KUKA KRL program: C2_CicloCompleto.src, C2_CicloCompleto.dat

--- C2_CicloCompleto.src ---
&ACCESS RVO1
&REL 253
&PARAM DISKPATH = KRC:\R1\Program\Work
DEF  C2_CicloCompleto (limpieza:IN)
   BOOL bTornillo, limpieza
   DECL INT velocidadAnterior,contadorPasadasLaser
   ;FOLD PROGRAM INFO --------------------------------------------------------
      ; Program: C2_CicloCompleto
      ; Description:
      ; Creation Date: 16/04/2024
      ; Last Modification Date: 14/09/2025
      ; Author:
      ;           Alexander Kalis
      ;           Tekniker, C. Iñaki Goenaga, 5, 20600, Gipuzkoa
      ;           +34 674 05 15 10
      ;           alexander.kalis@tekniker.es
      ; Last modification Author:
      ;           Alexander Kalis
      ; Customer: Erreka S. COOP
   ;ENDFOLD --------------------------------------------------------

   ;FOLD INI;%{PE}
      ;FOLD BASISTECH INI
         GLOBAL INTERRUPT DECL 3 WHEN $STOPMESS==TRUE DO IR_STOPM ( )
         INTERRUPT ON 3
         BAS (#INITMOV,0 )
      ;ENDFOLD (BASISTECH INI)

      ;FOLD USER INI
         ;Make your modifications here
         bTornillo=$IN[139]
         contadorPasadasLaser=0
         ;laserFrames = posCalcLaserSweep($RECIPE, $LAYOUT)
         ;laserFrames = posCalcLaserSweepAngledP($RECIPE, $LAYOUT, 5)
         laserFrames = posCalcLaserSweepAngledN($RECIPE, $LAYOUT, angle_barrido_laserAB)

         ;paintFrames = posCalcPaintSweep($RECIPE, $LAYOUT)
         ;paintFrames = posCalcPaintSweepAngledP($RECIPE, $LAYOUT, 5)
         paintFrames = posCalcPaintSweepAngledN($RECIPE, $LAYOUT, angle_barrido_pinturaAB)
      ;ENDFOLD (USER INI)
   ;ENDFOLD (INI)

   ;FOLD SPTP HOME CONT Vel=100 % DEFAULT ;%{PE}
      ;FOLD Parameters ;%{h}
         ;Params IlfProvider=kukaroboter.basistech.inlineforms.movement.spline; Kuka.IsGlobalPoint=False; Kuka.PointName=HOME; Kuka.BlendingEnabled=True; Kuka.MoveDataPtpName=DEFAULT; Kuka.VelocityPtp=100; Kuka.VelocityFieldEnabled=True; Kuka.ColDetectFieldEnabled=True; Kuka.CurrentCDSetIndex=0; Kuka.MovementParameterFieldEnabled=True; IlfCommand=SPTP
      ;ENDFOLD
      SPTP XHOME WITH $VEL_AXIS[1] = SVEL_JOINT(100.0), $TOOL = STOOL2(FHOME), $BASE = SBASE(FHOME.BASE_NO), $IPO_MODE = SIPO_MODE(FHOME.IPO_FRAME), $LOAD = SLOAD(FHOME.TOOL_NO), $ACC_AXIS[1] = SACC_JOINT(PDEFAULT), $APO = SAPO_PTP(PDEFAULT), $GEAR_JERK[1] = SGEAR_JERK(PDEFAULT), $COLLMON_TOL_PRO[1] = USE_CM_PRO_VALUES(0) C_Spl
   ;ENDFOLD

   ;FOLD Path to laser station
      IF limpieza THEN
         ;FOLD SPTP PTL1 CONT Vel=100 % PDAT13 Tool[1]:pintxoEstatico Base[2]:laserTCP extTCP  ;%{PE}
            ;FOLD Parameters ;%{h}
               ;Params IlfProvider=kukaroboter.basistech.inlineforms.movement.spline; Kuka.IsGlobalPoint=False; Kuka.PointName=PTL1; Kuka.BlendingEnabled=True; Kuka.MoveDataPtpName=PDAT13; Kuka.VelocityPtp=100; Kuka.VelocityFieldEnabled=True; Kuka.ColDetectFieldEnabled=True; Kuka.CurrentCDSetIndex=0; Kuka.MovementParameterFieldEnabled=True; IlfCommand=SPTP
            ;ENDFOLD
            SPTP XPTL1 WITH $VEL_AXIS[1] = SVEL_JOINT(100.0), $TOOL = STOOL2(FPTL1), $BASE = SBASE(FPTL1.BASE_NO), $IPO_MODE = SIPO_MODE(FPTL1.IPO_FRAME), $LOAD = SLOAD(FPTL1.TOOL_NO), $ACC_AXIS[1] = SACC_JOINT(PPDAT13), $APO = SAPO_PTP(PPDAT13), $GEAR_JERK[1] = SGEAR_JERK(PPDAT13), $COLLMON_TOL_PRO[1] = USE_CM_PRO_VALUES(0) C_Spl
         ;ENDFOLD
   ;ENDFOLD

   ;FOLD LASER PROCESS
      ;FOLD INIT barrido
         $TOOL = TOOL_DATA[1]
         $BASE = BASE_DATA[2]
         $IPO_MODE = #TCP
      ;ENDFOLD

      ;BUCLE DEPENDIENDO DEL NUMERO DE PASADAS

      ;FOLD Limpieza exterior esparrago
         $TOOL = TOOL_DATA[1] : laserFrames.screwBottom
         TRIGGER WHEN PATH = 0 ONSTART DELAY = 0 DO autMotorON() PRIO = 101
         TRIGGER WHEN PATH = 0 ONSTART DELAY = 0 DO autLaserON() PRIO = 102
         SPTP $NULLFRAME:C2LaserOffset[$RECIPE.recipeNum].sBO WITH $VEL.CP = laserParameter[$RECIPE.recipeNum].vel2, $VEL.ORI1 = laserParameter[$RECIPE.recipeNum].velRot2, $VEL.ORI2 = laserParameter[$RECIPE.recipeNum].velRot2
         WAIT SEC laserParameter[$RECIPE.recipeNum].tClean1
      ;ENDFOLD
      ;FOLD Limpieza perfil esparrago (punto A)
         $TOOL = TOOL_DATA[1] : laserFrames.screwProfileA
         SLIN $NULLFRAME:C2LaserOffset[$RECIPE.recipeNum].sPAO WITH $VEL.CP = laserParameter[$RECIPE.recipeNum].vel1, $VEL.ORI1 = laserParameter[$RECIPE.recipeNum].velRot1, $VEL.ORI2 = laserParameter[$RECIPE.recipeNum].velRot1
      ;ENDFOLD
      ;FOLD Limpieza perfil esparrago (punto B)
         velocidadAnterior = $OV_PRO
         $OV_PRO = 100
         $TOOL = TOOL_DATA[1] : laserFrames.screwProfileB
         SLIN $NULLFRAME:C2LaserOffset[$RECIPE.recipeNum].sPBO WITH $VEL.CP = laserParameter[$RECIPE.recipeNum].velSweep, $VEL.ORI1 = laserParameter[$RECIPE.recipeNum].velRot1, $VEL.ORI2 = laserParameter[$RECIPE.recipeNum].velRot1
         $OV_PRO = velocidadAnterior
      ;ENDFOLD
      contadorPasadasLaser=contadorPasadasLaser+1
      IF (bTornillo) THEN
         ;FOLD Limpieza perfil cabeza
            $TOOL = TOOL_DATA[1] : laserFrames.screwHex
            SLIN $NULLFRAME:C2LaserOffset[$RECIPE.recipeNum].sHO WITH $VEL.CP = laserParameter[$RECIPE.recipeNum].vel1, $VEL.ORI1 = laserParameter[$RECIPE.recipeNum].velRot1, $VEL.ORI2 = laserParameter[$RECIPE.recipeNum].velRot1
            WAIT SEC laserParameter[$RECIPE.recipeNum].tHex
         ;ENDFOLD
         ;FOLD Limpieza interior cabeza
            $TOOL = TOOL_DATA[1] : laserFrames.screwInnerHead
            SLIN $NULLFRAME:C2LaserOffset[$RECIPE.recipeNum].sIHO WITH $VEL.CP = laserParameter[$RECIPE.recipeNum].vel1, $VEL.ORI1 = laserParameter[$RECIPE.recipeNum].velRot1, $VEL.ORI2 = laserParameter[$RECIPE.recipeNum].velRot1
            WAIT SEC laserParameter[$RECIPE.recipeNum].tClean2
         ;ENDFOLD
      ENDIF

      ;FOLD Limpieza exterior cabeza
         $TOOL = TOOL_DATA[1] : laserFrames.screwOuterHead
         SLIN $NULLFRAME:C2LaserOffset[$RECIPE.recipeNum].sOHO WITH $VEL.CP = laserParameter[$RECIPE.recipeNum].vel1, $VEL.ORI1 = laserParameter[$RECIPE.recipeNum].velRot1, $VEL.ORI2 = laserParameter[$RECIPE.recipeNum].velRot1
         WAIT SEC laserParameter[$RECIPE.recipeNum].tClean3
      ;ENDFOLD
      ;Vuelta con angulo negativo B->A
      WHILE (ByNPasadasLaser > contadorPasadasLaser)
         ;FOLD Limpieza perfil esparrago (punto B)
            $TOOL = TOOL_DATA[1] : laserFrames.screwProfileB
            SLIN $NULLFRAME:C2LaserOffset[$RECIPE.recipeNum].sPBO WITH $VEL.CP = laserParameter[$RECIPE.recipeNum].vel1, $VEL.ORI1 = laserParameter[$RECIPE.recipeNum].velRot1, $VEL.ORI2 = laserParameter[$RECIPE.recipeNum].velRot1
         ;ENDFOLD
         ;FOLD Limpieza perfil esparrago (punto A)
            $TOOL = TOOL_DATA[1] : laserFrames.screwProfileA
            SLIN $NULLFRAME:C2LaserOffset[$RECIPE.recipeNum].sPAO WITH $VEL.CP = laserParameter[$RECIPE.recipeNum].velSweep, $VEL.ORI1 = laserParameter[$RECIPE.recipeNum].velRot1, $VEL.ORI2 = laserParameter[$RECIPE.recipeNum].velRot1
         ;ENDFOLD
         contadorPasadasLaser = contadorPasadasLaser + 1
      ENDWHILE
      autLaserOFF()
      autMotorOff()
      ENDIF
         ;ENDFOLD


   ;FOLD Path to DRYZONE
      petitionPermission(bPetEntradaLamparas, bPermisoEntradaLamparas)
   ;ENDFOLD

   ;FOLD Path to Paint station
      ;FOLD SPTP LTP1 CONT Vel=100 % PDAT17 Tool[1]:pintxoEstatico Base[3]:pintura ;%{PE}
         ;FOLD Parameters ;%{h}
            ;Params IlfProvider=kukaroboter.basistech.inlineforms.movement.spline; Kuka.IsGlobalPoint=False; Kuka.PointName=LTP1; Kuka.BlendingEnabled=True; Kuka.MoveDataPtpName=PDAT17; Kuka.VelocityPtp=100; Kuka.VelocityFieldEnabled=True; Kuka.ColDetectFieldEnabled=True; Kuka.CurrentCDSetIndex=0; Kuka.MovementParameterFieldEnabled=True; IlfCommand=SPTP
         ;ENDFOLD
         SPTP XLTP1 WITH $VEL_AXIS[1] = SVEL_JOINT(100.0), $TOOL = STOOL2(FLTP1), $BASE = SBASE(FLTP1.BASE_NO), $IPO_MODE = SIPO_MODE(FLTP1.IPO_FRAME), $LOAD = SLOAD(FLTP1.TOOL_NO), $ACC_AXIS[1] = SACC_JOINT(PPDAT17), $APO = SAPO_PTP(PPDAT17), $GEAR_JERK[1] = SGEAR_JERK(PPDAT17), $COLLMON_TOL_PRO[1] = USE_CM_PRO_VALUES(0) C_Spl
      ;ENDFOLD

   ;ENDFOLD

   ;FOLD PAINT PROCESS

      ;FOLD INIT barrido
         $TOOL = TOOL_DATA[1]
         $BASE = BASE_DATA[3]
         $IPO_MODE = #TCP
      ;ENDFOLD

      ;FOLD Pintado exterior esparrago
         TRIGGER WHEN PATH = 0 DELAY = 0 DO autPaintON() PRIO = 108
         TRIGGER WHEN PATH = 0 ONSTART DELAY = 0 DO autMotorOn() PRIO = 109
         $TOOL = TOOL_DATA[1] : paintFrames.screwBottom
         SPTP $NULLFRAME WITH $VEL.CP = paintParameter[$RECIPE.recipeNum].vel2, $VEL.ORI1 = paintParameter[$RECIPE.recipeNum].velRot2, $VEL.ORI2 = paintParameter[$RECIPE.recipeNum].velRot2
         WAIT SEC paintParameter[$RECIPE.recipeNum].tPaint1
         TRIGGER WHEN PATH = 0 ONSTART DELAY = 0 DO autPaintOFF() PRIO = 110
      ;ENDFOLD
      ;FOLD Pintado perfil esparrago (punto A)
         velocidadAnterior = $OV_PRO
         $TOOL = TOOL_DATA[1] : paintFrames.screwProfileA
         TRIGGER WHEN PATH = 0 DELAY = 0 DO autPaintON() PRIO = 111

         SLIN $NULLFRAME WITH $VEL.CP = paintParameter[$RECIPE.recipeNum].vel1, $VEL.ORI1 = paintParameter[$RECIPE.recipeNum].velRot1, $VEL.ORI2 = paintParameter[$RECIPE.recipeNum].velRot1
         $OV_PRO = 100
      ;ENDFOLD
      ;FOLD Pintado perfil esparrago (punto B)
         $TOOL = TOOL_DATA[1] : paintFrames.screwProfileB
         SLIN $NULLFRAME  WITH $VEL.CP = paintParameter[$RECIPE.recipeNum].velSweep, $VEL.ORI1 = paintParameter[$RECIPE.recipeNum].velRot1, $VEL.ORI2 = paintParameter[$RECIPE.recipeNum].velRot1
         TRIGGER WHEN PATH = 0 ONSTART DELAY = 0 DO autPaintOFF() PRIO = 112
         $OV_PRO = velocidadAnterior
      ;ENDFOLD
      IF (bTornillo) THEN
         ;FOLD Pintado perfil cabeza
            $TOOL = TOOL_DATA[1] : paintFrames.screwHex
            SLIN $NULLFRAME  WITH $VEL.CP = paintParameter[$RECIPE.recipeNum].vel1, $VEL.ORI1 = paintParameter[$RECIPE.recipeNum].velRot1, $VEL.ORI2 = paintParameter[$RECIPE.recipeNum].velRot1
            TRIGGER WHEN PATH = 0 DELAY = 0 DO autPaintON() PRIO = 113
            WAIT SEC paintParameter[$RECIPE.recipeNum].tHex
            TRIGGER WHEN PATH = 0 ONSTART DELAY = 0 DO autPaintOFF() PRIO = 114
         ;ENDFOLD
         ;FOLD Pintado interior cabeza
            TRIGGER WHEN PATH = 0 DELAY = 0 DO autPaintON() PRIO = 115
            $TOOL = TOOL_DATA[1] : paintFrames.screwInnerHead
            SLIN $NULLFRAME  WITH $VEL.CP = paintParameter[$RECIPE.recipeNum].vel1, $VEL.ORI1 = paintParameter[$RECIPE.recipeNum].velRot1, $VEL.ORI2 = paintParameter[$RECIPE.recipeNum].velRot1
            WAIT SEC paintParameter[$RECIPE.recipeNum].tPaint2
            TRIGGER WHEN PATH = 0 ONSTART DELAY = 0 DO autPaintOFF() PRIO = 116
         ;ENDFOLD
      ENDIF
      ;FOLD Pintado exterior cabeza
         $TOOL = TOOL_DATA[1] : paintFrames.screwOuterHead
         TRIGGER WHEN PATH = 0 DELAY = 0 DO autPaintON() PRIO = 117
         SPTP $NULLFRAME WITH $VEL.CP = paintParameter[$RECIPE.recipeNum].vel1, $VEL.ORI1 = paintParameter[$RECIPE.recipeNum].velRot1, $VEL.ORI2 = paintParameter[$RECIPE.recipeNum].velRot1
         WAIT SEC paintParameter[$RECIPE.recipeNum].tPaint3
         TRIGGER WHEN PATH = 0 ONSTART DELAY = 0 DO autPaintOFF() PRIO = 118
         autLamaparasOn()
      ;ENDFOLD

   ;ENDFOLD

   dryPos = posCalcDry($RECIPE, $LAYOUT)

   ;FOLD Path to wait Zone
;FOLD SPTP p10 CONT Vel=100 % PDAT19 Tool[1]:pintxoEstatico Base[4]:lamparas ;%{PE}
;FOLD Parameters ;%{h}
;Params IlfProvider=kukaroboter.basistech.inlineforms.movement.spline; Kuka.IsGlobalPoint=False; Kuka.PointName=p10; Kuka.BlendingEnabled=True; Kuka.MoveDataPtpName=PDAT19; Kuka.VelocityPtp=100; Kuka.VelocityFieldEnabled=True; Kuka.ColDetectFieldEnabled=True; Kuka.CurrentCDSetIndex=0; Kuka.MovementParameterFieldEnabled=True; IlfCommand=SPTP
;ENDFOLD
SPTP Xp10 WITH $VEL_AXIS[1] = SVEL_JOINT(100.0), $TOOL = STOOL2(Fp10), $BASE = SBASE(Fp10.BASE_NO), $IPO_MODE = SIPO_MODE(Fp10.IPO_FRAME), $LOAD = SLOAD(Fp10.TOOL_NO), $ACC_AXIS[1] = SACC_JOINT(PPDAT19), $APO = SAPO_PTP(PPDAT19), $GEAR_JERK[1] = SGEAR_JERK(PPDAT19), $COLLMON_TOL_PRO[1] = USE_CM_PRO_VALUES(0) C_Spl
;ENDFOLD
;FOLD SPTP p11 CONT Vel=100 % PDAT21 Tool[1]:pintxoEstatico Base[3]:pintura ;%{PE}
;FOLD Parameters ;%{h}
;Params IlfProvider=kukaroboter.basistech.inlineforms.movement.spline; Kuka.IsGlobalPoint=False; Kuka.PointName=p11; Kuka.BlendingEnabled=True; Kuka.MoveDataPtpName=PDAT21; Kuka.VelocityPtp=100; Kuka.VelocityFieldEnabled=True; Kuka.ColDetectFieldEnabled=True; Kuka.CurrentCDSetIndex=0; Kuka.MovementParameterFieldEnabled=True; IlfCommand=SPTP
;ENDFOLD
SPTP Xp11 WITH $VEL_AXIS[1] = SVEL_JOINT(100.0), $TOOL = STOOL2(Fp11), $BASE = SBASE(Fp11.BASE_NO), $IPO_MODE = SIPO_MODE(Fp11.IPO_FRAME), $LOAD = SLOAD(Fp11.TOOL_NO), $ACC_AXIS[1] = SACC_JOINT(PPDAT21), $APO = SAPO_PTP(PPDAT21), $GEAR_JERK[1] = SGEAR_JERK(PPDAT21), $COLLMON_TOL_PRO[1] = USE_CM_PRO_VALUES(0) C_Spl
;ENDFOLD
;FOLD SPTP p12 CONT Vel=100 % PDAT20 Tool[1]:pintxoEstatico Base[4]:lamparas ;%{PE}
;FOLD Parameters ;%{h}
;Params IlfProvider=kukaroboter.basistech.inlineforms.movement.spline; Kuka.IsGlobalPoint=False; Kuka.PointName=p12; Kuka.BlendingEnabled=True; Kuka.MoveDataPtpName=PDAT20; Kuka.VelocityPtp=100; Kuka.VelocityFieldEnabled=True; Kuka.ColDetectFieldEnabled=True; Kuka.CurrentCDSetIndex=0; Kuka.MovementParameterFieldEnabled=True; IlfCommand=SPTP
;ENDFOLD
SPTP Xp12 WITH $VEL_AXIS[1] = SVEL_JOINT(100.0), $TOOL = STOOL2(Fp12), $BASE = SBASE(Fp12.BASE_NO), $IPO_MODE = SIPO_MODE(Fp12.IPO_FRAME), $LOAD = SLOAD(Fp12.TOOL_NO), $ACC_AXIS[1] = SACC_JOINT(PPDAT20), $APO = SAPO_PTP(PPDAT20), $GEAR_JERK[1] = SGEAR_JERK(PPDAT20), $COLLMON_TOL_PRO[1] = USE_CM_PRO_VALUES(0) C_Spl
;ENDFOLD

   ;ENDFOLD

   ;FOLD Drying Process
      ;FOLD INIT barrido
         $TOOL = TOOL_DATA[1]
         $BASE = BASE_DATA[4]
         $IPO_MODE = #BASE

      ;ENDFOLD
      SLIN dryPos:dryAppOffset C_SPL
      SLIN dryPos WITH $VEL.CP = 3
      WAIT SEC tiempoSecado
      autMotorOff()
      autLamparasOff()
      SLIN dryPos:dryAppOffset C_DIS
   ;ENDFOLD

   ;FOLD Place Process
      petitionPermission(bPetEntradaDejarIND, bPermisoEntradaIND)

      ;FOLD INIT place
         $TOOL             =  TOOL_DATA[1]
         $BASE             =  BASE_DATA[5]
         placePos          =  $NULLPOS : posCalcPlaceIND($RECIPE, $LAYOUT)
         placeYOffset.Y    =  -5
      ;ENDFOLD

      SLIN placePos : mechanicalOffset : $RECIPE.PlO                     ;Punto de dejada
      autGripperOpen()
      SLIN placePos : placeYOffset : mechanicalOffset : $RECIPE.PlO       ;Punto de dejada con movimiento lateral
      SLIN_REL {Z 300}  C_SPL
   ;ENDFOLD

   ;FOLD Path to home

   ;ENDFOLD

   ;FOLD SPTP HOME Vel=100 % DEFAULT ;%{PE}
      ;FOLD Parameters ;%{h}
         ;Params IlfProvider=kukaroboter.basistech.inlineforms.movement.spline; Kuka.IsGlobalPoint=False; Kuka.PointName=HOME; Kuka.BlendingEnabled=False; Kuka.MoveDataPtpName=DEFAULT; Kuka.VelocityPtp=100; Kuka.VelocityFieldEnabled=True; Kuka.CurrentCDSetIndex=0; Kuka.MovementParameterFieldEnabled=True; IlfCommand=SPTP
      ;ENDFOLD
      SPTP XHOME WITH $VEL_AXIS[1] = SVEL_JOINT(100.0), $TOOL = STOOL2(FHOME), $BASE = SBASE(FHOME.BASE_NO), $IPO_MODE = SIPO_MODE(FHOME.IPO_FRAME), $LOAD = SLOAD(FHOME.TOOL_NO), $ACC_AXIS[1] = SACC_JOINT(PDEFAULT), $APO = SAPO_PTP(PDEFAULT), $GEAR_JERK[1] = SGEAR_JERK(PDEFAULT), $COLLMON_TOL_PRO[1] = USE_CM_PRO_VALUES(0)
   ;ENDFOLD

END

--- C2_CicloCompleto.dat ---
&ACCESS RVO1
&REL 253
&PARAM DISKPATH = KRC:\R1\Program\Work
DEFDAT  C2_CICLOCOMPLETO
;FOLD EXTERNAL DECLARATIONS;%{PE}%MKUKATPBASIS,%CEXT,%VCOMMON,%P
;FOLD BASISTECH EXT;%{PE}%MKUKATPBASIS,%CEXT,%VEXT,%P
EXT  BAS (BAS_COMMAND  :IN,REAL  :IN )
DECL INT SUCCESS
;ENDFOLD (BASISTECH EXT)
;FOLD USER EXT;%{E}%MKUKATPUSER,%CEXT,%VEXT,%P
;Make your modifications here

;ENDFOLD (USER EXT)
;ENDFOLD (EXTERNAL DECLARATIONS)

;--------------
DECL laserSweepFrames laserFrames
DECL laserSweepFrames paintFrames

DECL POS dryPos={X -28.0000,Y -675.000,Z 0.0,A 0.0,B 0.0,C 0.0,S 0,T 0}
DECL POS placePos={X 0.0,Y -567.000,Z 31.7512875,A 0.0,B 0.0,C 0.0}
DECL FRAME placeYOffset={X 0.0,Y -5.00000,Z 0.0,A 0.0,B 0.0,C 0.0}
DECL FRAME dryAppOffset={X -250.000,Y 0.0,Z -25.0000,A 0.0,B 0.0,C 0.0}
DECL FRAME mechanicalOffset={X 0.0,Y 0.0,Z 0.0,A 0.0,B 0.0,C 0.0}
;--------------

DECL MODULEPARAM_T LAST_TP_PARAMS={PARAMS[] "Kuka.Logics.Io=1; Kuka.Logics.IoName=; Kuka.Logics.State=True; Kuka.Logics.Cont=False; Kuka.Logics.Time=0.1; Kuka.VelocityFieldEnabled=True; Kuka.ColDetectFieldEnabled=True; Kuka.MovementParameterFieldEnabled=True; Kuka.IsAngleEnabled=False; Kuka.PointName=p12; Kuka.FrameData.base_no=4; Kuka.FrameData.tool_no=1; Kuka.FrameData.ipo_frame=#BASE; Kuka.isglobalpoint=False; Kuka.MoveDataPtpName=PDAT20; Kuka.MovementDataPdat.apo_mode=#CDIS; Kuka.MovementDataPdat.apo_dist=500; Kuka.MovementData.vel=100; Kuka.MovementData.acc=100; Kuka.MovementData.exax_ign=0; Kuka.VelocityPtp=100; Kuka.BlendingEnabled=True; Kuka.APXEnabled=False; Kuka.CurrentCDSetIndex=0; Kuka.FrameData.point2=; Kuka.MoveDataName=CPDAT3; Kuka.MovementData.cb={AUX_PT {ORI #CONSIDER,E1 #CONSIDER,E2 #CONSIDER,E3 #CONSIDER,E4 #CONSIDER,E5 #CONSIDER,E6 #CONSIDER},TARGET_PT {ORI #INTERPOLATE,E1 #INTERPOLATE,E2 #INTERPOLATE,E3 #INTERPOLATE,E4 #INTERPOLATE,E5 #INTERPOLATE,E6 #INTERPOLATE}}; Kuka.MovementData.apo_fac=50; Kuka.MovementData.apo_dist=500; Kuka.MovementData.axis_acc=100; Kuka.MovementData.axis_vel=100; Kuka.MovementData.circ_typ=#BASE; Kuka.MovementData.jerk_fac=50; Kuka.MovementData.ori_typ=#VAR; Kuka.VelocityPath=2  "}
DECL E6POS Xp1={X 32.6300697,Y -469.728973,Z -186.153549,A 0.0174859129,B -0.00349956797,C 0.00372947869,S 22,T 51,E1 0.0,E2 0.0,E3 0.0,E4 0.0,E5 0.0,E6 0.0}
DECL FDAT Fp1={TOOL_NO 1,BASE_NO 2,IPO_FRAME #TCP,POINT2[] " "}
DECL PDAT PPDAT1={VEL 100.000,ACC 100.000,APO_DIST 500.000,APO_MODE #CDIS,GEAR_JERK 100.000,EXAX_IGN 0}
DECL E6POS Xp2={X 1604.48621,Y 119.015739,Z 987.622314,A -49.9389381,B -0.0320644975,C -0.0134176081,S 18,T 34,E1 0.0,E2 0.0,E3 0.0,E4 0.0,E5 0.0,E6 0.0}
DECL FDAT Fp2={TOOL_NO 1,BASE_NO 0,IPO_FRAME #BASE,POINT2[] " "}
DECL PDAT PPDAT2={VEL 100.000,ACC 100.000,APO_DIST 500.000,APO_MODE #CDIS,GEAR_JERK 100.000,EXAX_IGN 0}
DECL E6POS Xp3={X 1604.76404,Y 118.793060,Z 1122.24011,A -49.9511948,B -0.0349329337,C -0.0147130266,S 18,T 34,E1 0.0,E2 0.0,E3 0.0,E4 0.0,E5 0.0,E6 0.0}
DECL FDAT Fp3={TOOL_NO 1,BASE_NO 0,IPO_FRAME #BASE,POINT2[] " "}
DECL PDAT PPDAT3={VEL 100.000,ACC 100.000,APO_DIST 500.000,APO_MODE #CDIS,GEAR_JERK 100.000,EXAX_IGN 0}
DECL E6POS Xp4={X 11.3002872,Y -327.049713,Z 1.53383017,A 0.0190707371,B -0.000264858070,C -0.000815795793,S 22,T 51,E1 0.0,E2 0.0,E3 0.0,E4 0.0,E5 0.0,E6 0.0}
DECL FDAT Fp4={TOOL_NO 1,BASE_NO 2,IPO_FRAME #TCP,POINT2[] " "}
DECL PDAT PPDAT4={VEL 100.000,ACC 100.000,APO_DIST 500.000,APO_MODE #CDIS,GEAR_JERK 100.000,EXAX_IGN 0}
DECL E6POS Xp5={X 28.2340622,Y -18.8887100,Z -412.324615,A -3.73290348,B -0.0232962687,C 0.0178582016,S 22,T 50,E1 0.0,E2 0.0,E3 0.0,E4 0.0,E5 0.0,E6 0.0}
DECL FDAT Fp5={TOOL_NO 1,BASE_NO 2,IPO_FRAME #TCP,POINT2[] " "}
DECL PDAT PPDAT5={VEL 100.000,ACC 100.000,APO_DIST 500.000,APO_MODE #CDIS,GEAR_JERK 100.000,EXAX_IGN 0}
DECL E6POS Xp6={X 28.2340622,Y -18.8887100,Z -412.324615,A -3.73290348,B -0.0232962687,C 0.0178582016,S 22,T 50,E1 0.0,E2 0.0,E3 0.0,E4 0.0,E5 0.0,E6 0.0}
DECL FDAT Fp6={TOOL_NO 1,BASE_NO 2,IPO_FRAME #TCP,POINT2[] " "}
DECL PDAT PPDAT6={VEL 100.000,ACC 100.000,APO_DIST 500.000,APO_MODE #CDIS,GEAR_JERK 100.000,EXAX_IGN 0}
DECL E6POS Xp7={X 590.350037,Y -636.649414,Z -415.669403,A -0.136172593,B -0.156493708,C -0.0280757807,S 22,T 50,E1 0.0,E2 0.0,E3 0.0,E4 0.0,E5 0.0,E6 0.0}
DECL FDAT Fp7={TOOL_NO 1,BASE_NO 2,IPO_FRAME #TCP,POINT2[] " "}
DECL PDAT PPDAT7={VEL 100.000,ACC 100.000,APO_DIST 500.000,APO_MODE #CDIS,GEAR_JERK 100.000,EXAX_IGN 0}
DECL E6POS Xp8={X -1455.58374,Y 237.404190,Z -275.962891,A 144.069733,B 4.96351290,C 0.0175147261,S 18,T 34,E1 0.0,E2 0.0,E3 0.0,E4 0.0,E5 0.0,E6 0.0}
DECL FDAT Fp8={TOOL_NO 1,BASE_NO 2,IPO_FRAME #TCP,POINT2[] " "}
DECL LDAT LCPDAT1={VEL 2.00000,ACC 100.000,APO_DIST 500.000,APO_FAC 50.0000,AXIS_VEL 100.000,AXIS_ACC 100.000,ORI_TYP #VAR,CIRC_TYP #BASE,JERK_FAC 50.0000,GEAR_JERK 100.000,EXAX_IGN 0,CB {AUX_PT {ORI #CONSIDER,E1 #CONSIDER,E2 #CONSIDER,E3 #CONSIDER,E4 #CONSIDER,E5 #CONSIDER,E6 #CONSIDER},TARGET_PT {ORI #INTERPOLATE,E1 #INTERPOLATE,E2 #INTERPOLATE,E3 #INTERPOLATE,E4 #INTERPOLATE,E5 #INTERPOLATE,E6 #INTERPOLATE}}}
DECL E6POS Xp9={X 666666.688,Y 66.6000,Z 666.660,A 6.60000,B 66.6600,C 666.600,S 0,T 0,E1 0.0,E2 0.0,E3 0.0,E4 0.0,E5 0.0,E6 0.0}
DECL FDAT Fp9={TOOL_NO 1,BASE_NO 2,IPO_FRAME #TCP,POINT2[] " "}
DECL LDAT LCPDAT2={VEL 2.00000,ACC 100.000,APO_DIST 500.000,APO_FAC 50.0000,AXIS_VEL 100.000,AXIS_ACC 100.000,ORI_TYP #VAR,CIRC_TYP #BASE,JERK_FAC 50.0000,GEAR_JERK 100.000,EXAX_IGN 0,CB {AUX_PT {ORI #CONSIDER,E1 #CONSIDER,E2 #CONSIDER,E3 #CONSIDER,E4 #CONSIDER,E5 #CONSIDER,E6 #CONSIDER},TARGET_PT {ORI #INTERPOLATE,E1 #INTERPOLATE,E2 #INTERPOLATE,E3 #INTERPOLATE,E4 #INTERPOLATE,E5 #INTERPOLATE,E6 #INTERPOLATE}}}
DECL E6POS Xp10={X -704.420715,Y 696.612122,Z 327.585449,A -3.93213654,B 24.0421619,C -4.06740332,S 18,T 34,E1 0.0,E2 0.0,E3 0.0,E4 0.0,E5 0.0,E6 0.0}
DECL FDAT Fp10={TOOL_NO 1,BASE_NO 4,IPO_FRAME #BASE,POINT2[] " "}
DECL PDAT PPDAT8={VEL 100.000,ACC 100.000,APO_DIST 500.000,APO_MODE #CDIS,GEAR_JERK 100.000,EXAX_IGN 0}

DECL PDAT PPDAT9={VEL 100.000,ACC 100.000,APO_DIST 500.000,APO_MODE #CDIS,GEAR_JERK 100.000,EXAX_IGN 0}
DECL E6POS Xpaint1={X -41.2740135,Y -822.688477,Z 2.95846963,A -40.1920204,B -4.24734831,C 2.30867672,S 18,T 43,E1 0.0,E2 0.0,E3 0.0,E4 0.0,E5 0.0,E6 0.0}
DECL FDAT Fpaint1={TOOL_NO 1,BASE_NO 3,IPO_FRAME #TCP,POINT2[] " "}
DECL PDAT PPDAT10={VEL 100.000,ACC 100.000,APO_DIST 500.000,APO_MODE #CDIS,GEAR_JERK 100.000,EXAX_IGN 0}
DECL E6POS Xpait2={X -104.701454,Y -113.430878,Z -20.5580807,A -9.25399590,B -4.45930529,C -0.106951475,S 18,T 42,E1 0.0,E2 0.0,E3 0.0,E4 0.0,E5 0.0,E6 0.0}
DECL FDAT Fpait2={TOOL_NO 1,BASE_NO 3,IPO_FRAME #TCP,POINT2[] " "}
DECL PDAT PPDAT11={VEL 100.000,ACC 100.000,APO_DIST 500.000,APO_MODE #CDIS,GEAR_JERK 100.000,EXAX_IGN 0}
DECL E6POS Xpait3={X -84.4007568,Y 241.647430,Z -23.1614609,A 1.55418110,B -3.23597527,C -0.101248451,S 18,T 42,E1 0.0,E2 0.0,E3 0.0,E4 0.0,E5 0.0,E6 0.0}
DECL FDAT Fpait3={TOOL_NO 1,BASE_NO 3,IPO_FRAME #TCP,POINT2[] " "}
DECL PDAT PPDAT12={VEL 100.000,ACC 100.000,APO_DIST 500.000,APO_MODE #CDIS,GEAR_JERK 100.000,EXAX_IGN 0}
DECL E6POS Xhtl1={X -553.719788,Y -2125.48560,Z -497.483368,A -70.8249664,B 0.133065462,C 0.103076503,S 18,T 35,E1 0.0,E2 0.0,E3 0.0,E4 0.0,E5 0.0,E6 0.0}
DECL FDAT Fhtl1={TOOL_NO 1,BASE_NO 3,IPO_FRAME #TCP,POINT2[] " "}
DECL PDAT PPDAT13={VEL 100.000,ACC 100.000,APO_DIST 200.000,APO_MODE #CDIS,GEAR_JERK 100.000,EXAX_IGN 0}
DECL E6POS XPTL1={X -279.476929,Y 221.876572,Z -289.029449,A 9.12497425,B 0.00512073468,C -0.193030745,S 18,T 43,E1 0.0,E2 0.0,E3 0.0,E4 0.0,E5 0.0,E6 0.0}
DECL FDAT FPTL1={TOOL_NO 1,BASE_NO 2,IPO_FRAME #TCP,POINT2[] " "}
DECL E6POS XPTP1={X 21.1799145,Y -1107.35425,Z -12.1308088,A -1.84557688,B -0.228079408,C 0.451393425,S 18,T 43,E1 0.0,E2 0.0,E3 0.0,E4 0.0,E5 0.0,E6 0.0}
DECL FDAT FPTP1={TOOL_NO 1,BASE_NO 3,IPO_FRAME #TCP,POINT2[] " "}
DECL PDAT PPDAT14={VEL 100.000,ACC 100.000,APO_DIST 100.000,APO_MODE #CDIS,GEAR_JERK 100.000,EXAX_IGN 0}
DECL E6POS XLTP1={X 39.1310158,Y 1219.16907,Z 3.74033594,A 4.72046089,B 0.263525456,C -0.468695700,S 18,T 43,E1 0.0,E2 0.0,E3 0.0,E4 0.0,E5 0.0,E6 0.0}
DECL FDAT FLTP1={TOOL_NO 1,BASE_NO 3,IPO_FRAME #BASE,POINT2[] " "}
DECL PDAT PPDAT15={VEL 100.000,ACC 100.000,APO_DIST 200.000,APO_MODE #CDIS,GEAR_JERK 100.000,EXAX_IGN 0}
DECL E6POS XLTP2={X -525.198181,Y 1217.20789,Z 9.22105503,A 0.0868065804,B -0.227606848,C -0.232948631,S 18,T 43,E1 0.0,E2 0.0,E3 0.0,E4 0.0,E5 0.0,E6 0.0}
DECL FDAT FLTP2={TOOL_NO 1,BASE_NO 2,IPO_FRAME #TCP,POINT2[] " "}
DECL PDAT PPDAT16={VEL 100.000,ACC 100.000,APO_DIST 200.000,APO_MODE #CDIS,GEAR_JERK 100.000,EXAX_IGN 0}
DECL PDAT PPDAT17={VEL 100.000,ACC 100.000,APO_DIST 200.000,APO_MODE #CDIS,GEAR_JERK 100.000,EXAX_IGN 0}
DECL E6POS Xp11={X -1713.32410,Y -1255.66040,Z 691.988647,A -86.8421326,B -30.1441727,C -0.373799175,S 18,T 10,E1 0.0,E2 0.0,E3 0.0,E4 0.0,E5 0.0,E6 0.0}
DECL FDAT Fp11={TOOL_NO 1,BASE_NO 3,IPO_FRAME #BASE,POINT2[] " "}
DECL PDAT PPDAT18={VEL 50.0000,ACC 100.000,APO_DIST 200.000,APO_MODE #CDIS,GEAR_JERK 100.000,EXAX_IGN 0}
DECL LDAT LCPDAT3={VEL 2.00000,ACC 100.000,APO_DIST 500.000,APO_FAC 50.0000,AXIS_VEL 100.000,AXIS_ACC 100.000,ORI_TYP #VAR,CIRC_TYP #BASE,JERK_FAC 50.0000,GEAR_JERK 100.000,EXAX_IGN 0,CB {AUX_PT {ORI #CONSIDER,E1 #CONSIDER,E2 #CONSIDER,E3 #CONSIDER,E4 #CONSIDER,E5 #CONSIDER,E6 #CONSIDER},TARGET_PT {ORI #INTERPOLATE,E1 #INTERPOLATE,E2 #INTERPOLATE,E3 #INTERPOLATE,E4 #INTERPOLATE,E5 #INTERPOLATE,E6 #INTERPOLATE}}}
DECL PDAT PPDAT19={VEL 100.000,ACC 100.000,APO_DIST 500.000,APO_MODE #CDIS,GEAR_JERK 100.000,EXAX_IGN 0}
DECL E6POS Xp12={X -268.007172,Y -1099.99951,Z -25.0012379,A 1.47648907E-05,B 0.000233355488,C 5.48213757E-05,S 18,T 10,E1 0.0,E2 0.0,E3 0.0,E4 0.0,E5 0.0,E6 0.0}
DECL FDAT Fp12={TOOL_NO 1,BASE_NO 4,IPO_FRAME #BASE,POINT2[] " "}
DECL PDAT PPDAT20={VEL 100.000,ACC 100.000,APO_DIST 500.000,APO_MODE #CDIS,GEAR_JERK 100.000,EXAX_IGN 0}
DECL PDAT PPDAT21={VEL 100.000,ACC 100.000,APO_DIST 500.000,APO_MODE #CDIS,GEAR_JERK 100.000,EXAX_IGN 0}
ENDDAT
